TYPE VelocityCtrl_Output_typ :
	STRUCT
		monitor 	: Velocityctrl_monitor_typ ;
		Status		: VelocityCtrl_Status_typ ;
		Error		: VelocityCtrl_Error_typ ;
		
	END_STRUCT
END_TYPE

(* stored: Version 1.1.0.1, ProductVersion 3.1.4024.3
   DUT VelocityCtrl_Output_typ: Id {e6ade8fb-a66a-43e5-896d-10d75ca507eb} *)
